Staubli VAL3: ReadHead.pgx

program ReadHead(num x_nFileID, bool& x_bHeaderOk, string& x_sPrdID, tool& x_tTool, joint& x_jHome, frame& x_fFrame, trsf& x_trOffset, num& x_nTotalTrajs)
  local num l_nRead
  local string l_sRead
  local num l_nFind
  local string l_sSplit[2]
  local string l_sValue[10]
  local bool b[7]
begin

  nFileId=$fileOpen(sFileName,"r")
  if nFileId>=0 and nFileId<=9
    x_bHeaderOk=false
    while !x_bHeaderOk
      l_nRead=$fileGet(nFileId,l_sRead,1)
      //
      call split(l_sRead,"=",l_sSplit)
      if l_sSplit[1]=="BEGIN"
        x_bHeaderOk=true
        return
      endIf

      call split(l_sSplit[1],",",l_sValue)



      //
      switch l_sSplit[0]
        case "PRODUCTID"
          x_sPrdID=l_sValue[0]
        break
        case "TOOL"
          l_sValue[0]=toNum(l_sValue[0],x_tTool.trsf.x,b[1])
          l_sValue[1]=toNum(l_sValue[1],x_tTool.trsf.y,b[2])
          l_sValue[2]=toNum(l_sValue[2],x_tTool.trsf.z,b[3])
          l_sValue[3]=toNum(l_sValue[3],x_tTool.trsf.rx,b[4])
          l_sValue[4]=toNum(l_sValue[4],x_tTool.trsf.ry,b[5])
          l_sValue[5]=toNum(l_sValue[5],x_tTool.trsf.rz,b[6])
        break
        case "HOME"
          l_sValue[0]=toNum(l_sValue[0],x_jHome.j1,b[1])
          l_sValue[1]=toNum(l_sValue[1],x_jHome.j2,b[2])
          l_sValue[2]=toNum(l_sValue[2],x_jHome.j3,b[3])
          l_sValue[3]=toNum(l_sValue[3],x_jHome.j4,b[4])
          l_sValue[4]=toNum(l_sValue[4],x_jHome.j5,b[5])
          l_sValue[5]=toNum(l_sValue[5],x_jHome.j6,b[6])
        break
        case "FRAME"
          l_sValue[0]=toNum(l_sValue[0],x_fFrame.trsf.x,b[1])
          l_sValue[1]=toNum(l_sValue[1],x_fFrame.trsf.y,b[2])
          l_sValue[2]=toNum(l_sValue[2],x_fFrame.trsf.z,b[3])
          l_sValue[3]=toNum(l_sValue[3],x_fFrame.trsf.rx,b[4])
          l_sValue[4]=toNum(l_sValue[4],x_fFrame.trsf.ry,b[5])
          l_sValue[5]=toNum(l_sValue[5],x_fFrame.trsf.rz,b[6])
        break
        case "OFFSET"
          l_sValue[0]=toNum(l_sValue[0],x_trOffset.x,b[1])
          l_sValue[1]=toNum(l_sValue[1],x_trOffset.y,b[2])
          l_sValue[2]=toNum(l_sValue[2],x_trOffset.z,b[3])
          l_sValue[3]=toNum(l_sValue[3],x_trOffset.rx,b[4])
          l_sValue[4]=toNum(l_sValue[4],x_trOffset.ry,b[5])
          l_sValue[5]=toNum(l_sValue[5],x_trOffset.rz,b[6])
        break
        case "TOTALTRAJS"
          l_sValue[0]=toNum(l_sValue[0],x_nTotalTrajs,b[1])
        break
      endSwitch
      //当提取到=后面的"BEGIN"时,头文件读取结束

    endWhile
  else
    popUpMsg(sFileName+"does not open")
    logMsg(sFileName+"does not open")
    x_bHeaderOk=false
  endIf

end
